ABB RAPID module: 002A09EA

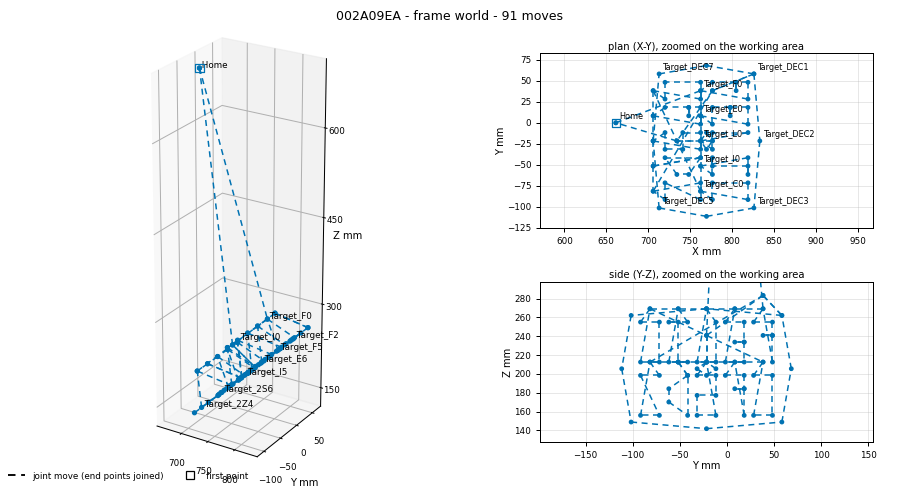
[picture p0: tool path of 002A09EA in frame world, 91 of 91 moves have a stored position in this frame; points joined in program order, loops and branches not executed]
MODULE Module1
        PERS tooldata Marcador:=[TRUE,[[25.287,0,146.409],[0.996194698,0,0.087155743,0]],[0.1,[0,0,1],[1,0,0,0],0,0,0]];
    TASK PERS wobjdata WO_Pastel:=[FALSE,TRUE,"",[[833.258893819,68.374306775,269.142643333],[0,-0.382683433,0,0.923879532]],[[0,0,0],[1,0,0,0]]];
    CONST robtarget Target_F0:=[[50,30,50],[0,0,1,0],[0,0,0,0],[9E+09,9E+09,9E+09,9E+09,9E+09,9E+09]];
    CONST robtarget Target_F1:=[[20,20,0],[0,0,1,0],[0,0,0,0],[9E+09,9E+09,9E+09,9E+09,9E+09,9E+09]];
    CONST robtarget Target_F2:=[[20,40,0],[0,0,1,0],[0,0,0,0],[9E+09,9E+09,9E+09,9E+09,9E+09,9E+09]];
    CONST robtarget Target_F3:=[[40,20,0],[0,0,1,0],[0,0,0,0],[9E+09,9E+09,9E+09,9E+09,9E+09,9E+09]];
    CONST robtarget Target_F4:=[[40,30,0],[0,0,1,0],[0,0,0,0],[9E+09,9E+09,9E+09,9E+09,9E+09,9E+09]];
    CONST robtarget Target_F5:=[[80,20,0],[0,0,1,0],[0,0,0,0],[9E+09,9E+09,9E+09,9E+09,9E+09,9E+09]];
    CONST robtarget Target_E0:=[[50,60,50],[0,0,1,0],[0,0,0,0],[9E+09,9E+09,9E+09,9E+09,9E+09,9E+09]];
    CONST robtarget Target_E1:=[[20,50,0],[0,0,1,0],[0,0,0,0],[9E+09,9E+09,9E+09,9E+09,9E+09,9E+09]];
    CONST robtarget Target_E2:=[[20,70,0],[0,0,1,0],[0,0,0,0],[9E+09,9E+09,9E+09,9E+09,9E+09,9E+09]];
    CONST robtarget Target_E3:=[[50,50,0],[0,0,1,0],[0,0,0,0],[9E+09,9E+09,9E+09,9E+09,9E+09,9E+09]];
    CONST robtarget Target_E4:=[[50,60,0],[0,0,1,0],[0,0,0,0],[9E+09,9E+09,9E+09,9E+09,9E+09,9E+09]];
    CONST robtarget Target_E5:=[[80,50,0],[0,0,1,0],[0,0,0,0],[9E+09,9E+09,9E+09,9E+09,9E+09,9E+09]];
    CONST robtarget Target_E6:=[[80,70,0],[0,0,1,0],[0,0,0,0],[9E+09,9E+09,9E+09,9E+09,9E+09,9E+09]];
    CONST robtarget Target_L0:=[[50,90,50],[0,0,1,0],[0,0,0,0],[9E+09,9E+09,9E+09,9E+09,9E+09,9E+09]];
    CONST robtarget Target_L1:=[[20,80,0],[0,0,1,0],[0,0,0,0],[9E+09,9E+09,9E+09,9E+09,9E+09,9E+09]];
    CONST robtarget Target_L2:=[[80,80,0],[0,0,1,0],[0,0,0,0],[9E+09,9E+09,9E+09,9E+09,9E+09,9E+09]];
    CONST robtarget Target_L3:=[[80,100,0],[0,0,1,0],[0,0,0,0],[9E+09,9E+09,9E+09,9E+09,9E+09,9E+09]];
    CONST robtarget Target_I0:=[[50,120,50],[0,0,1,0],[0,0,0,0],[9E+09,9E+09,9E+09,9E+09,9E+09,9E+09]];
    CONST robtarget Target_I1:=[[20,110,0],[0,0,1,0],[0,0,0,0],[9E+09,9E+09,9E+09,9E+09,9E+09,9E+09]];
    CONST robtarget Target_I2:=[[20,120,0],[0,0,1,0],[0,0,0,0],[9E+09,9E+09,9E+09,9E+09,9E+09,9E+09]];
    CONST robtarget Target_I3:=[[20,130,0],[0,0,1,0],[0,0,0,0],[9E+09,9E+09,9E+09,9E+09,9E+09,9E+09]];
    CONST robtarget Target_I4:=[[80,110,0],[0,0,1,0],[0,0,0,0],[9E+09,9E+09,9E+09,9E+09,9E+09,9E+09]];
    CONST robtarget Target_I5:=[[80,120,0],[0,0,1,0],[0,0,0,0],[9E+09,9E+09,9E+09,9E+09,9E+09,9E+09]];
    CONST robtarget Target_I6:=[[80,130,0],[0,0,1,0],[0,0,0,0],[9E+09,9E+09,9E+09,9E+09,9E+09,9E+09]];
    CONST robtarget Target_C0:=[[50,150,50],[0,0,1,0],[0,0,0,0],[9E+09,9E+09,9E+09,9E+09,9E+09,9E+09]];
    CONST robtarget Target_C1:=[[20,140,0],[0,0,1,0],[0,0,0,0],[9E+09,9E+09,9E+09,9E+09,9E+09,9E+09]];
    CONST robtarget Target_C2:=[[20,160,0],[0,0,1,0],[0,0,0,0],[9E+09,9E+09,9E+09,9E+09,9E+09,9E+09]];
    CONST robtarget Target_C3:=[[80,140,0],[0,0,1,0],[0,0,0,0],[9E+09,9E+09,9E+09,9E+09,9E+09,9E+09]];
    CONST robtarget Target_C4:=[[80,160,0],[0,0,1,0],[0,0,0,0],[9E+09,9E+09,9E+09,9E+09,9E+09,9E+09]];
    CONST robtarget Target_2C0:=[[130,30,50],[0,0,1,0],[0,0,0,0],[9E+09,9E+09,9E+09,9E+09,9E+09,9E+09]];
    CONST robtarget Target_2C1:=[[100,20,0],[0,0,1,0],[0,0,0,0],[9E+09,9E+09,9E+09,9E+09,9E+09,9E+09]];
    CONST robtarget Target_2C2:=[[100,40,0],[0,0,1,0],[0,0,0,0],[9E+09,9E+09,9E+09,9E+09,9E+09,9E+09]];
    CONST robtarget Target_2C3:=[[160,20,0],[0,0,1,0],[0,0,0,0],[9E+09,9E+09,9E+09,9E+09,9E+09,9E+09]];
    CONST robtarget Target_2C4:=[[160,40,0],[0,0,1,0],[0,0,0,0],[9E+09,9E+09,9E+09,9E+09,9E+09,9E+09]];
    CONST robtarget Target_2F0:=[[130,60,50],[0,0,1,0],[0,0,0,0],[9E+09,9E+09,9E+09,9E+09,9E+09,9E+09]];
    CONST robtarget Target_2F1:=[[100,50,0],[0,0,1,0],[0,0,0,0],[9E+09,9E+09,9E+09,9E+09,9E+09,9E+09]];
    CONST robtarget Target_2F2:=[[100,70,0],[0,0,1,0],[0,0,0,0],[9E+09,9E+09,9E+09,9E+09,9E+09,9E+09]];
    CONST robtarget Target_2F3:=[[120,50,0],[0,0,1,0],[0,0,0,0],[9E+09,9E+09,9E+09,9E+09,9E+09,9E+09]];
    CONST robtarget Target_2F4:=[[120,60,0],[0,0,1,0],[0,0,0,0],[9E+09,9E+09,9E+09,9E+09,9E+09,9E+09]];
    CONST robtarget Target_2F5:=[[160,50,0],[0,0,1,0],[0,0,0,0],[9E+09,9E+09,9E+09,9E+09,9E+09,9E+09]];
    CONST robtarget Target_2S0:=[[130,90,50],[0,0,1,0],[0,0,0,0],[9E+09,9E+09,9E+09,9E+09,9E+09,9E+09]];
    CONST robtarget Target_2S1:=[[100,80,0],[0,0,1,0],[0,0,0,0],[9E+09,9E+09,9E+09,9E+09,9E+09,9E+09]];
    CONST robtarget Target_2S2:=[[100,100,0],[0,0,1,0],[0,0,0,0],[9E+09,9E+09,9E+09,9E+09,9E+09,9E+09]];
    CONST robtarget Target_2S3:=[[130,80,0],[0,0,1,0],[0,0,0,0],[9E+09,9E+09,9E+09,9E+09,9E+09,9E+09]];
    CONST robtarget Target_2S4:=[[130,100,0],[0,0,1,0],[0,0,0,0],[9E+09,9E+09,9E+09,9E+09,9E+09,9E+09]];
    CONST robtarget Target_2S5:=[[160,80,0],[0,0,1,0],[0,0,0,0],[9E+09,9E+09,9E+09,9E+09,9E+09,9E+09]];
    CONST robtarget Target_2S6:=[[160,100,0],[0,0,1,0],[0,0,0,0],[9E+09,9E+09,9E+09,9E+09,9E+09,9E+09]];
    CONST robtarget Target_2D0:=[[130,120,50],[0,0,1,0],[0,0,0,0],[9E+09,9E+09,9E+09,9E+09,9E+09,9E+09]];
    CONST robtarget Target_2D1:=[[100,110,0],[0,0,1,0],[0,0,0,0],[9E+09,9E+09,9E+09,9E+09,9E+09,9E+09]];
    CONST robtarget Target_2D2:=[[120,130,0],[0,0,1,0],[0,0,0,0],[9E+09,9E+09,9E+09,9E+09,9E+09,9E+09]];
    CONST robtarget Target_2D3:=[[140,130,0],[0,0,1,0],[0,0,0,0],[9E+09,9E+09,9E+09,9E+09,9E+09,9E+09]];
    CONST robtarget Target_2D4:=[[160,110,0],[0,0,1,0],[0,0,0,0],[9E+09,9E+09,9E+09,9E+09,9E+09,9E+09]];
    CONST robtarget Target_2Z0:=[[130,150,50],[0,0,1,0],[0,0,0,0],[9E+09,9E+09,9E+09,9E+09,9E+09,9E+09]];
    CONST robtarget Target_2Z1:=[[100,140,0],[0,0,1,0],[0,0,0,0],[9E+09,9E+09,9E+09,9E+09,9E+09,9E+09]];
    CONST robtarget Target_2Z2:=[[100,160,0],[0,0,1,0],[0,0,0,0],[9E+09,9E+09,9E+09,9E+09,9E+09,9E+09]];
    CONST robtarget Target_2Z3:=[[160,140,0],[0,0,1,0],[0,0,0,0],[9E+09,9E+09,9E+09,9E+09,9E+09,9E+09]];
    CONST robtarget Target_2Z4:=[[160,160,0],[0,0,1,0],[0,0,0,0],[9E+09,9E+09,9E+09,9E+09,9E+09,9E+09]];
    CONST robtarget Target_DEC0:=[[30,30,50],[0,0,1,0],[0,0,0,0],[9E+09,9E+09,9E+09,9E+09,9E+09,9E+09]];
    CONST robtarget Target_DEC1:=[[10,10,0],[0,0,1,0],[0,0,0,0],[9E+09,9E+09,9E+09,9E+09,9E+09,9E+09]];
    CONST robtarget Target_DEC2:=[[0,90,0],[0,0,1,0],[0,0,0,0],[9E+09,9E+09,9E+09,9E+09,9E+09,9E+09]];
    CONST robtarget Target_DEC3:=[[10,170,0],[0,0,1,0],[0,0,0,0],[9E+09,9E+09,9E+09,9E+09,9E+09,9E+09]];
    CONST robtarget Target_DEC4:=[[90,180,0],[0,0,1,0],[0,0,0,0],[9E+09,9E+09,9E+09,9E+09,9E+09,9E+09]];
    CONST robtarget Target_DEC5:=[[170,170,0],[0,0,1,0],[0,0,0,0],[9E+09,9E+09,9E+09,9E+09,9E+09,9E+09]];
    CONST robtarget Target_DEC6:=[[180,90,0],[0,0,1,0],[0,0,0,0],[9E+09,9E+09,9E+09,9E+09,9E+09,9E+09]];
    CONST robtarget Target_DEC7:=[[170,10,0],[0,0,1,0],[0,0,0,0],[9E+09,9E+09,9E+09,9E+09,9E+09,9E+09]];
    CONST robtarget Target_DEC8:=[[90,0,0],[0,0,1,0],[0,0,0,0],[9E+09,9E+09,9E+09,9E+09,9E+09,9E+09]];
    CONST robtarget Target_2DEC0:=[[90,90,50],[0,0,1,0],[0,0,0,0],[9E+09,9E+09,9E+09,9E+09,9E+09,9E+09]];
    CONST robtarget Target_2DEC1:=[[80,90,0],[0,0,1,0],[0,0,0,0],[9E+09,9E+09,9E+09,9E+09,9E+09,9E+09]];
    CONST robtarget Target_2DEC2:=[[90,100,0],[0,0,1,0],[0,0,0,0],[9E+09,9E+09,9E+09,9E+09,9E+09,9E+09]];
    CONST robtarget Target_2DEC3:=[[100,90,0],[0,0,1,0],[0,0,0,0],[9E+09,9E+09,9E+09,9E+09,9E+09,9E+09]];
    CONST robtarget Target_2DEC4:=[[90,80,0],[0,0,1,0],[0,0,0,0],[9E+09,9E+09,9E+09,9E+09,9E+09,9E+09]];
    CONST robtarget Home:=[[661.409,0,686.713],[0.642787609,0,0.766044443,0],[0,0,0,0],[9E+09,9E+09,9E+09,9E+09,9E+09,9E+09]];
!***********************************************************
    !
    ! Módulo:  Module1
    !
    ! Descripción:
    !   <Introduzca la descripción aquí>
    !
    ! Autor: felip
    !
    ! Versión: 1.0
    !
    !***********************************************************


    !***********************************************************
    !
    ! Procedimiento Main
    !
    !   Este es el punto de entrada de su programa
    !
    !***********************************************************
    PROC main()
        !Añada aquí su código
        Path_10;
    ENDPROC
    PROC Path_10()
        MoveJ Home,v100,z100,Marcador\WObj:=wobj0;
        MoveJ Target_F0,v100,fine,Marcador\WObj:=WO_Pastel;
        MoveJ Target_F2,v100,fine,Marcador\WObj:=WO_Pastel;
        MoveJ Target_F1,v100,fine,Marcador\WObj:=WO_Pastel;
        MoveJ Target_F3,v100,fine,Marcador\WObj:=WO_Pastel;
        MoveJ Target_F4,v100,fine,Marcador\WObj:=WO_Pastel;
        MoveJ Target_F3,v100,fine,Marcador\WObj:=WO_Pastel;
        MoveJ Target_F5,v100,fine,Marcador\WObj:=WO_Pastel;
        MoveJ Target_F0,v100,fine,Marcador\WObj:=WO_Pastel;
        MoveJ Target_E0,v100,fine,Marcador\WObj:=WO_Pastel;
        MoveJ Target_E2,v100,fine,Marcador\WObj:=WO_Pastel;
        MoveJ Target_E1,v100,fine,Marcador\WObj:=WO_Pastel;
        MoveJ Target_E3,v100,fine,Marcador\WObj:=WO_Pastel;
        MoveJ Target_E4,v100,fine,Marcador\WObj:=WO_Pastel;
        MoveJ Target_E3,v100,fine,Marcador\WObj:=WO_Pastel;
        MoveJ Target_E5,v100,fine,Marcador\WObj:=WO_Pastel;
        MoveJ Target_E6,v100,fine,Marcador\WObj:=WO_Pastel;
        MoveJ Target_E0,v100,fine,Marcador\WObj:=WO_Pastel;
        MoveJ Target_L0,v100,fine,Marcador\WObj:=WO_Pastel;
        MoveJ Target_L1,v100,fine,Marcador\WObj:=WO_Pastel;
        MoveJ Target_L2,v100,fine,Marcador\WObj:=WO_Pastel;
        MoveJ Target_L3,v100,fine,Marcador\WObj:=WO_Pastel;
        MoveJ Target_L0,v100,fine,Marcador\WObj:=WO_Pastel;
        MoveJ Target_I0,v100,fine,Marcador\WObj:=WO_Pastel;
        MoveJ Target_I1,v100,fine,Marcador\WObj:=WO_Pastel;
        MoveJ Target_I3,v100,fine,Marcador\WObj:=WO_Pastel;
        MoveJ Target_I2,v100,fine,Marcador\WObj:=WO_Pastel;
        MoveJ Target_I5,v100,fine,Marcador\WObj:=WO_Pastel;
        MoveJ Target_I4,v100,fine,Marcador\WObj:=WO_Pastel;
        MoveJ Target_I6,v100,fine,Marcador\WObj:=WO_Pastel;
        MoveJ Target_I0,v100,fine,Marcador\WObj:=WO_Pastel;
        MoveJ Target_C0,v100,fine,Marcador\WObj:=WO_Pastel;
        MoveJ Target_C2,v100,fine,Marcador\WObj:=WO_Pastel;
        MoveJ Target_C1,v100,fine,Marcador\WObj:=WO_Pastel;
        MoveJ Target_C3,v100,fine,Marcador\WObj:=WO_Pastel;
        MoveJ Target_C4,v100,fine,Marcador\WObj:=WO_Pastel;
        MoveJ Target_C0,v100,fine,Marcador\WObj:=WO_Pastel;
        MoveJ Target_2C0,v100,fine,Marcador\WObj:=WO_Pastel;
        MoveJ Target_2C2,v100,fine,Marcador\WObj:=WO_Pastel;
        MoveJ Target_2C1,v100,fine,Marcador\WObj:=WO_Pastel;
        MoveJ Target_2C3,v100,fine,Marcador\WObj:=WO_Pastel;
        MoveJ Target_2C4,v100,fine,Marcador\WObj:=WO_Pastel;
        MoveJ Target_2C0,v100,fine,Marcador\WObj:=WO_Pastel;
        MoveJ Target_2F0,v100,fine,Marcador\WObj:=WO_Pastel;
        MoveJ Target_2F2,v100,fine,Marcador\WObj:=WO_Pastel;
        MoveJ Target_2F1,v100,fine,Marcador\WObj:=WO_Pastel;
        MoveJ Target_2F3,v100,fine,Marcador\WObj:=WO_Pastel;
        MoveJ Target_2F4,v100,fine,Marcador\WObj:=WO_Pastel;
        MoveJ Target_2F3,v100,fine,Marcador\WObj:=WO_Pastel;
        MoveJ Target_2F5,v100,fine,Marcador\WObj:=WO_Pastel;
        MoveJ Target_2F0,v100,fine,Marcador\WObj:=WO_Pastel;
        MoveJ Target_2S0,v100,fine,Marcador\WObj:=WO_Pastel;
        MoveJ Target_2S2,v100,fine,Marcador\WObj:=WO_Pastel;
        MoveJ Target_2S1,v100,fine,Marcador\WObj:=WO_Pastel;
        MoveJ Target_2S3,v100,fine,Marcador\WObj:=WO_Pastel;
        MoveJ Target_2S4,v100,fine,Marcador\WObj:=WO_Pastel;
        MoveJ Target_2S6,v100,fine,Marcador\WObj:=WO_Pastel;
        MoveJ Target_2S5,v100,fine,Marcador\WObj:=WO_Pastel;
        MoveJ Target_2S0,v100,fine,Marcador\WObj:=WO_Pastel;
        MoveJ Target_2D0,v100,fine,Marcador\WObj:=WO_Pastel;
        MoveJ Target_2D1,v100,fine,Marcador\WObj:=WO_Pastel;
        MoveJ Target_2D2,v100,fine,Marcador\WObj:=WO_Pastel;
        MoveJ Target_2D3,v100,fine,Marcador\WObj:=WO_Pastel;
        MoveJ Target_2D4,v100,fine,Marcador\WObj:=WO_Pastel;
        MoveJ Target_2D1,v100,fine,Marcador\WObj:=WO_Pastel;
        MoveJ Target_2D0,v100,fine,Marcador\WObj:=WO_Pastel;
        MoveJ Target_2Z0,v100,fine,Marcador\WObj:=WO_Pastel;
        MoveJ Target_2Z1,v100,fine,Marcador\WObj:=WO_Pastel;
        MoveJ Target_2Z2,v100,fine,Marcador\WObj:=WO_Pastel;
        MoveJ Target_2Z3,v100,fine,Marcador\WObj:=WO_Pastel;
        MoveJ Target_2Z4,v100,fine,Marcador\WObj:=WO_Pastel;
        MoveJ Target_2Z0,v100,fine,Marcador\WObj:=WO_Pastel;
        MoveJ Target_DEC0,v100,fine,Marcador\WObj:=WO_Pastel;
        MoveJ Target_DEC1,v100,fine,Marcador\WObj:=WO_Pastel;
        MoveJ Target_DEC2,v100,fine,Marcador\WObj:=WO_Pastel;
        MoveJ Target_DEC3,v100,fine,Marcador\WObj:=WO_Pastel;
        MoveJ Target_DEC4,v100,fine,Marcador\WObj:=WO_Pastel;
        MoveJ Target_DEC5,v100,fine,Marcador\WObj:=WO_Pastel;
        MoveJ Target_DEC6,v100,fine,Marcador\WObj:=WO_Pastel;
        MoveJ Target_DEC7,v100,fine,Marcador\WObj:=WO_Pastel;
        MoveJ Target_DEC8,v100,fine,Marcador\WObj:=WO_Pastel;
        MoveJ Target_DEC1,v100,fine,Marcador\WObj:=WO_Pastel;
        MoveJ Target_DEC0,v100,fine,Marcador\WObj:=WO_Pastel;
        MoveJ Target_2DEC0,v100,fine,Marcador\WObj:=WO_Pastel;
        MoveJ Target_2DEC1,v100,fine,Marcador\WObj:=WO_Pastel;
        MoveJ Target_2DEC2,v100,fine,Marcador\WObj:=WO_Pastel;
        MoveJ Target_2DEC3,v100,fine,Marcador\WObj:=WO_Pastel;
        MoveJ Target_2DEC4,v100,fine,Marcador\WObj:=WO_Pastel;
        MoveJ Target_2DEC1,v100,fine,Marcador\WObj:=WO_Pastel;
        MoveJ Target_2DEC0,v100,fine,Marcador\WObj:=WO_Pastel;
        MoveJ Home,v100,z100,Marcador\WObj:=wobj0;
    ENDPROC
ENDMODULE
